FUNCTION_BLOCK EmergencyDecideInit2 (* Basic Function Block Type *)
  (* Standard: 61499-2 *)
  (* Version 0.0, 7/15/2026, Schneider Electric, Template *)
  PACKAGE SE.Nereda;
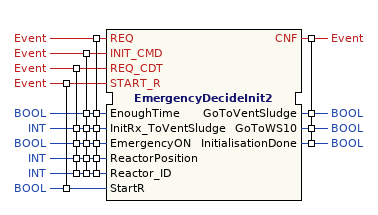
  EVENT_INPUT
    REQ WITH EnoughTime, InitRx_ToVentSludge, Reactor_ID, EmergencyON, ReactorPosition; (* Normal Execution Request *)
    INIT_CMD WITH EmergencyON, EnoughTime, InitRx_ToVentSludge, Reactor_ID, ReactorPosition;
    REQ_CDT WITH InitRx_ToVentSludge, Reactor_ID, EmergencyON, ReactorPosition;
    START_R WITH StartR;
  END_EVENT
  EVENT_OUTPUT
    CNF WITH GoToVentSludge, GoToWS10, InitialisationDone; (* Execution Confirmation *)
  END_EVENT
  VAR_INPUT
    EnoughTime : BOOL; (* Input event qualifier *)
    InitRx_ToVentSludge : INT;
    EmergencyON : BOOL;
    ReactorPosition : INT;
    Reactor_ID : INT;
    StartR : BOOL;
  END_VAR
  VAR_OUTPUT
    GoToVentSludge : BOOL; (* Output event qualifier *)
    GoToWS10 : BOOL;
    InitialisationDone : BOOL;
  END_VAR
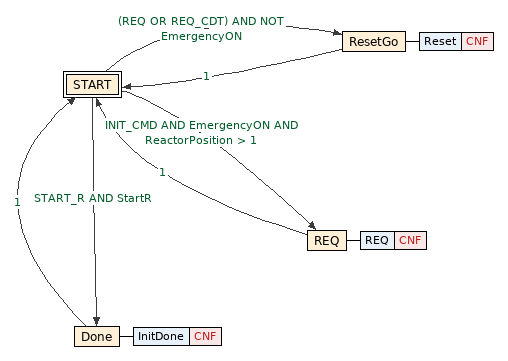
  EC_STATES
    START; (* Initial State *)
    REQ : REQ -> CNF; (* Normal execution *)
    ResetGo : Reset -> CNF;
    Done : InitDone -> CNF;
  END_STATES
  EC_TRANSITIONS
    START TO REQ := INIT_CMD AND EmergencyON AND ReactorPosition > 1;
    REQ TO START := 1;
    START TO ResetGo := (REQ OR REQ_CDT) AND NOT EmergencyON;
    ResetGo TO START := 1;
    START TO Done := START_R AND StartR;
    Done TO START := 1;
  END_TRANSITIONS
  ALGORITHM REQ IN ST: (* Normally executed algorithm *)
IF EnoughTime THEN
	GoToWS10 := FALSE;
	InitialisationDone := FALSE;
	IF InitRx_ToVentSludge = Reactor_ID THEN
		GoToVentSludge := TRUE;
		GoToWS10 := FALSE;
	END_IF;
ELSE
	GoToVentSludge := FALSE;
	GoToWS10 := TRUE;
	InitialisationDone := FALSE;
END_IF;
  END_ALGORITHM
  ALGORITHM Reset IN ST:
GoToVentSludge := FALSE;
GoToWS10 := FALSE;
  END_ALGORITHM
  ALGORITHM InitDone IN ST:
GoToVentSludge := FALSE;
GoToWS10 := FALSE;
InitialisationDone := TRUE;
  END_ALGORITHM
END_FUNCTION_BLOCK
